Yaskawa INFORM job: MTFTEST.JBI

/JOB
//NAME MTFTEST
//POS
///NPOS 0,0,0,0,0,0
//INST
///DATE 2024/01/24 13:09
///ATTR SC,RW,RJ
////FRAME ROBOT
///GROUP1 RB1,BS1
///LVARS 2,2,0,0,0,3,3,0
NOP
GETARG LI001 IARG#(1)
GETS LPX000 $PX016
CNVRT LPX000 LPX000 BF
SET LP001 P[LI001]
FOR LI000 START= 1 TO 3
	 SET LB000 LI000
	 SETE LP000 (LB000) 0
NEXT LI000
FOR LI000 START= 4 TO 6
	 SET LB000 LI000
	 SETE LP001 (LB000) 0
NEXT LI000
ADD LP000 LP001
SET P[LI001] LP000
END
